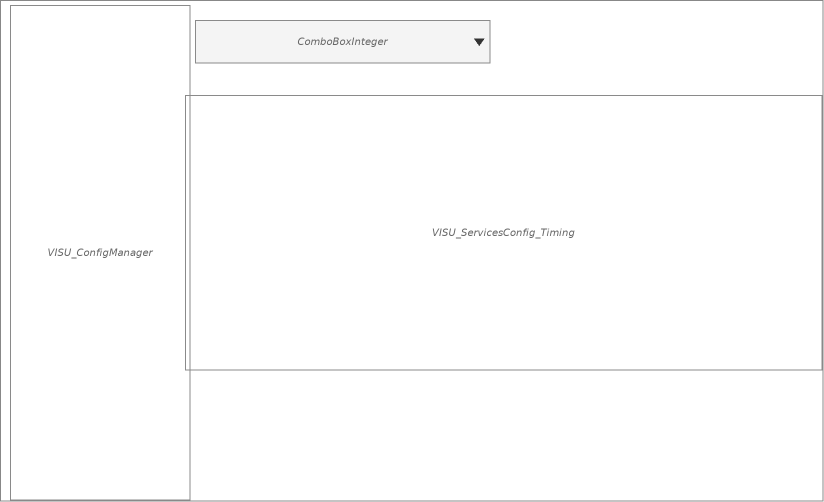
VISUALIZATION VISU_ServicesConfig  // 824x502
VAR_IN_OUT
    editableConfig : ServicesConfig;
	activeConfig : ServicesConfig;
    mgr : ConfigManager;
    mgrWidget : ConfigManagerWidget;
    activeTab : INT;
END_VAR
    Frame (10,5 180x495)
        shows VISU_ConfigManager(mgr := mgr, widget := mgrWidget)
    ComboBoxInteger (195,20 295x43), variable: activeTab, text list: 'ServicesConfigTabsTextList'
    Frame (185,95 637x275), frame switch variable: activeTab
        shows VISU_ServicesConfig_Timing(editableConfig := editableConfig.timing, activeConfig := activeConfig.timing)
END_VISUALIZATION

(* stored: Version 1.1.0.1, ProductVersion 3.1.4019.2
   Visu VISU_ServicesConfig: Id {1b1084c1-0edd-45fa-832e-e5daf7775e65} *)
